// TIA Portal V21 export
DATA_BLOCK "C0_ID"   // DB9
{ S7_Optimized_Access := 'TRUE' }
// stored: MemoryReserve 100
   VAR
      CabinetNumber : Int := 1;   // Current C0 cabinet to be programmed
   END_VAR
BEGIN
END_DATA_BLOCK
